FUNCTION_BLOCK FB_ValveBank IMPLEMENTS I_ValveBank
VAR_INPUT
	NumOfValves : INT;
END_VAR
VAR_OUTPUT
END_VAR
VAR
	aValves 	: ARRAY[1..NumOfValves] OF FB_Valve;
END_VAR

{warning 'add method implementation '}
METHOD AddValve : BOOL
END_METHOD

{warning 'add method implementation '}
METHOD GetValveStats : INT
END_METHOD

{warning 'add method implementation '}
METHOD TriggerFromMask : BOOL
VAR_INPUT
	aValveMask : ARRAY[1..NumOfValves] OF BOOL;
END_VAR
VAR
	i	: INT;
END_VAR
FOR i := 1 TO NumOfValves DO
	IF aVAlveMask[i] THEN
		aValves[i].CmdOpen();
	ELSE
		aValves[i].CmdClose();
	END_IF
END_FOR

TriggerFromMask := TRUE;
END_METHOD

END_FUNCTION_BLOCK

(* stored: Version 1.1.0.1, ProductVersion 3.1.4024.15
   POU FB_ValveBank: Id {6fd479d4-9175-4488-b2ec-fe7d4059738b}, SpecialFunc None
   Method AddValve: Id {3f4e104f-ebf9-455a-83e7-c19d6b83e420}
   Method GetValveStats: Id {a2aa7772-672a-422c-afc0-a68981b3618e}
   Method TriggerFromMask: Id {fe376a1d-db65-4f96-89c4-385f8cf1d130} *)
